{analysis '-23}
FUNCTION SYSTEM_TIME_TO_RFC3339 : STRING(255)
VAR_INPUT
	tCurrentTime	:	TIMESTRUCT;
END_VAR
VAR
END_VAR

SYSTEM_TIME_TO_RFC3339 := CONCAT(REPLACE(SYSTEMTIME_TO_STRING(tCurrentTime), 'T', 1, 11), 'Z');

END_FUNCTION

(* stored: Version 1.1.0.1, ProductVersion 3.1.4022.10
   POU SYSTEM_TIME_TO_RFC3339: Id {8224a586-2295-4f0e-ba2f-710d1a2cbe6b}, SpecialFunc None *)
